Fanuc KAREL source: kd00032.KL

-- PROVISIONAL review KL for V1013-1; original PC SHA256 e92d91e2a20f43d150f981fd70fe5c3823bcb238905a9a668cea49350e16710c
-- Incomplete behavior may be omitted. Consult companion uncertainty JSON. Do not deploy.
PROGRAM KD00032
%NOLOCKGROUP
VAR
  I : INTEGER
  J : INTEGER
  B : BOOLEAN
  R : REAL
  S : STRING[80]
BEGIN
  -- UNRESOLVED_PC offsets 5-25; opcodes 9D,81,18,2E,12,22,9D,13,04
  -- UNRESOLVED_PC offsets 30-34; opcodes 7F
END KD00032
